{attribute 'GeneratedUsingTerminal: IODEVICETYPE_ETHERCATPROT'}
{attribute addProperty BoxType "IODEVICETYPE_ETHERCATPROT"}
{attribute addProperty Id "Beckhoff_ER1xxxBeckhoff_ER1xxx_27EF5A30492Beckhoff_ER2xxxBeckhoff_ER2xxx_DC95CE44904Beckhoff_ER3xxxBeckhoff_ER3xxx_28EA77F5522Beckhoff_ER4xxxBeckhoff_ER4xxx_F39C275080Beckhoff_ER5xxxBeckhoff_ER5xxx_44A92E1E80Beckhoff_ER6xxxBeckhoff_ER6xxx_3F7F1EBD406Beckhoff_ER7xxxBeckhoff_ER7xxx_5C5227D6598Beckhoff_ER8xxxBeckhoff_ER8xxx_177550BF64SyncUnitsSyncUnits_99E584AF18InputsInputs_25A0042B160OutputsOutputs_2397A10E106InfoDataInfoData_C76BEFB322"}
{attribute addProperty CRC "2613864898"}
{attribute addProperty Size "3452"}
TYPE EtherCAT_Master_ERxxxx_9BCC69C2 :
STRUCT
	{attribute addProperty Name "Beckhoff_ER1xxx"}
	{attribute addProperty PreviousPort "EtherCAT_Master_ERxxxx : Master"}
	Beckhoff_ER1xxx : Beckhoff_ER1xxx_27EF5A30;
	{attribute addProperty Name "Beckhoff_ER2xxx"}
	{attribute addProperty PreviousPort "Beckhoff ER1xxx : C"}
	Beckhoff_ER2xxx : Beckhoff_ER2xxx_DC95CE44;
	{attribute addProperty Name "Beckhoff_ER3xxx"}
	{attribute addProperty PreviousPort "Beckhoff ER2xxx : C"}
	Beckhoff_ER3xxx : Beckhoff_ER3xxx_28EA77F5;
	{attribute addProperty Name "Beckhoff_ER4xxx"}
	{attribute addProperty PreviousPort "Beckhoff ER3xxx : C"}
	Beckhoff_ER4xxx : Beckhoff_ER4xxx_F39C2750;
	{attribute addProperty Name "Beckhoff_ER5xxx"}
	{attribute addProperty PreviousPort "Beckhoff ER4xxx : C"}
	Beckhoff_ER5xxx : Beckhoff_ER5xxx_44A92E1E;
	{attribute addProperty Name "Beckhoff_ER6xxx"}
	{attribute addProperty PreviousPort "Beckhoff ER5xxx : C"}
	Beckhoff_ER6xxx : Beckhoff_ER6xxx_3F7F1EBD;
	{attribute addProperty Name "Beckhoff_ER7xxx"}
	{attribute addProperty PreviousPort "Beckhoff ER6xxx : C"}
	Beckhoff_ER7xxx : Beckhoff_ER7xxx_5C5227D6;
	{attribute addProperty Name "Beckhoff_ER8xxx"}
	{attribute addProperty PreviousPort "Beckhoff ER7xxx : C"}
	Beckhoff_ER8xxx : Beckhoff_ER8xxx_177550BF;
	{attribute addProperty Name "SyncUnits"}
	SyncUnits : SyncUnits_99E584AF;
	{attribute addProperty Name "Inputs"}
	Inputs : Inputs_25A0042B;
	{attribute addProperty Name "Outputs"}
	Outputs : Outputs_2397A10E;
	{attribute addProperty Name "InfoData"}
	InfoData : InfoData_C76BEFB3;
END_STRUCT
END_TYPE

(* stored: Version 1.2.0.0, ProductVersion 3.1.4024.9
   DUT EtherCAT_Master_ERxxxx_9BCC69C2: Id {c69302c2-43b2-49bf-b94e-0587522d6d2a} *)
